(* PLC project actuator, TNI-Software ControlBuild 4.00.17 *)
(* stored: creationDateTime 2005-06-20T11:52:45-01:00 *)

FUNCTION_BLOCK cmd_equipment_library.actuator
  VAR_INPUT  (* CB.group=Modes CB.kind=inputVars *)
    autoMode : BOOL := false;  (* CB.mnemonicPatternPropertyName=<SY>_AUTO_<NU> CB.libelle=Automatic mode *)
    manualMode : BOOL := false;  (* CB.mnemonicPatternPropertyName=<SY>_MANU_<NU> CB.libelle=Manual mode *)
  END_VAR
  VAR_INPUT  (* CB.group=Commands CB.kind=inputVars *)
    autoFwdCmd : BOOL := false;  (* CB.mnemonicPatternPropertyName=<SY>_CMDFWAUTO_<NU> CB.libelle=Automatic forward command *)
    autoBwdCmd : BOOL := false;  (* CB.mnemonicPatternPropertyName=<SY>_CMDSAUTO_<NU> CB.libelle=Automatic backward command *)
  END_VAR
  VAR_INPUT  (* CB.group=PushButtons CB.kind=inputVars *)
    forwardPB : BOOL := false;  (* CB.mnemonicPatternPropertyName=<SY>_BPFW_<NU> CB.libelle=Forward pushbutton *)
    backwardPB : BOOL := false;  (* CB.mnemonicPatternPropertyName=<SY>_BPS_<NU> CB.libelle=Backward pushbutton *)
    offPB : BOOL := false;  (* CB.mnemonicPatternPropertyName=<SY>_BPARRET_<NU> CB.libelle=Off pushbutton *)
  END_VAR
  VAR_INPUT  (* CB.kind=inputVars *)
    generalFault : BOOL := false;  (* CB.mnemonicPatternPropertyName=<SY>_DEF_<NU> CB.libelle=General fault of the engine *)
  END_VAR
  VAR_OUTPUT  (* CB.group=Orders CB.kind=outputVars *)
    backwardCmd : BOOL := false;  (* CB.mnemonicPatternPropertyName=bwdCmd<SY><NU> CB.libelle=Backward command *)
    forwardCmd : BOOL := false;  (* CB.mnemonicPatternPropertyName=fwdCmd<SY><NU> CB.libelle=Forward command *)
  END_VAR

(* LD diagram, written out as Structured Text *)
1:
forwardCmd := (autoMode AND autoFwdCmd OR manualMode AND (forwardCmd OR forwardPB AND NOT backwardPB) AND NOT offPB AND NOT backwardCmd) AND NOT generalFault;
2:
backwardCmd := (autoMode AND autoBwdCmd OR manualMode AND (backwardCmd OR backwardPB AND NOT forwardPB) AND NOT offPB AND NOT forwardCmd) AND NOT generalFault;
END_FUNCTION_BLOCK
